{attribute 'qualified_only'}
VAR_GLOBAL
	axis_a : AXIS_REF;
END_VAR

(* stored: Version 1.1.0.1, ProductVersion 3.1.4024.12
   GVL GVL: Id {31be1bad-6f79-4db1-9bf7-219e70471568} *)
